
// ===== library: MasterCopy "UseCaseBasedDokuFB" =====

FUNCTION_BLOCK "UseCaseBasedDokuFB"   // FB4, FBD
TITLE = BasicFB
{ S7_Optimized_Access := 'TRUE' }
VERSION : 0.1
   VAR_INPUT
      Input1 : Bool;
      Input2 : Bool;
   END_VAR
   VAR_OUTPUT
      Output1 : Bool;
   END_VAR
BEGIN

REGION Network 1: AndNetwork1
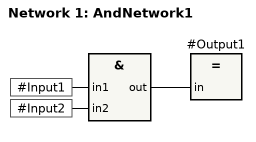
   #Output1 := #Input1 AND #Input2;
END_REGION
END_FUNCTION_BLOCK